// TIA Portal V19 export
DATA_BLOCK "CallEquipment_DB"   // DB107
AUTHOR : Siemens_FA_SUP
// stored: InstanceOfName Unit2.EM0.CallEquipment, InstanceOfType FB, Namespace Unit2.EM0
"Unit2.EM0.CallEquipment"
   // VAR_IN_OUT
   //    unitStatus : "LAF_typeUnitStatus";
   //    unitAlarmDB : "LAF_typeAlarms";
   //    emFeedback : "LUC_typeEmFeedback";
   // END_VAR
   // VAR
   //    statUnitStatus { ExternalWritable := 'False'} : "LAF_typeUnitStatus";
   //    instJob1 { ExternalWritable := 'False'} : "LAF_SelectJob";
   //    instSequence { ExternalWritable := 'False'} : "Unit2.EM0.Sequence";
   //    instManageBitAlarms { ExternalWritable := 'False'} : "LAF_ManageBitAlarms";
   // END_VAR
BEGIN
END_DATA_BLOCK
